ABB RobotStudio station: ExternalGuidedMotion.rsstn

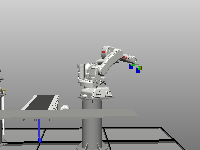
Station E459 (saved by RobotStudio format 3)
Controller NorbertEGMVirtual2, task T_ROB1: task frame (RAPID world) sits at (-305, -752, 720) mm, rotated rx 0 ry 0 rz 30 deg in the station
Controller NorbertEGMVirtual2
  mechanical unit ROB_1: Norbert, 6 joints, base frame (0, 0, 0) mm
  mechanical unit CNV1: ?, 1 joints, base frame (0, 0, 0) mm
Layout (positions relative to the parent item):
  - PedestalR [part, from Libraries\Pedestal.rslib] at (10, 680, 0) mm, rotated rx 0 ry 0 rz 150 deg
  - PedestalN [part, from Libraries\Pedestal.rslib] at (-305, -752, 0) mm, rotated rx 0 ry 0 rz -150 deg
  - Conveyor [part, from Libraries\Conveyor.rslib] at (-998.97, -64.27, 615.81) mm, rotated rx 90 ry 0 rz -90 deg
  - Windowtable [part]
  - BordR [part, from Libraries\Desk.rslib] at (193.4, 1497.66, 0) mm, rotated rx 0 ry 0 rz -120 deg
  - UISpenholder [mechanism, from Libraries\UISpenholder.rslib] at (483.21, 1099.62, 1138) mm, rotated rx -180 ry 0 rz 150 deg
  - Norbert [mechanism, from Robots\IRB140_6_81_C_G_03.rslib] at (-305, -752, 720) mm, rotated rx 0 ry 0 rz 30 deg; joint values [-1.5087, 0.9061, -0.6756, 0, 1.3403, 3.2037] (rad or m)
  - Rudolf [mechanism, from Robots\IRB140_6_81_C_G_03.rslib] at (10, 680, 720) mm, rotated rx 0 ry 0 rz -30 deg; joint values [1.249, 0.6446, -0.2193, 0, 1.1455, 1.249] (rad or m)
  - tSuctionCup [mechanism, from Libraries\tSuctionCup.rslib] at (94.83, -1354.75, 1142.25) mm, rotated rx -180 ry 0 rz -60 deg
Attachment: BordR is attached to PedestalR
Attachment: UISpenholder is attached to Rudolf / Link6
Attachment: tSuctionCup is attached to Norbert / Link6
Station signals: DI doClose, DI doOpen
Station logic (signal -> signal, property => property):
  NorbertEGMVirtual2.doOpen -> SC_Gripper.diOpen
  NorbertEGMVirtual2.doClose -> SC_Gripper.diClose
  SC_Gripper.doClosed -> NorbertEGMVirtual2.diClosed
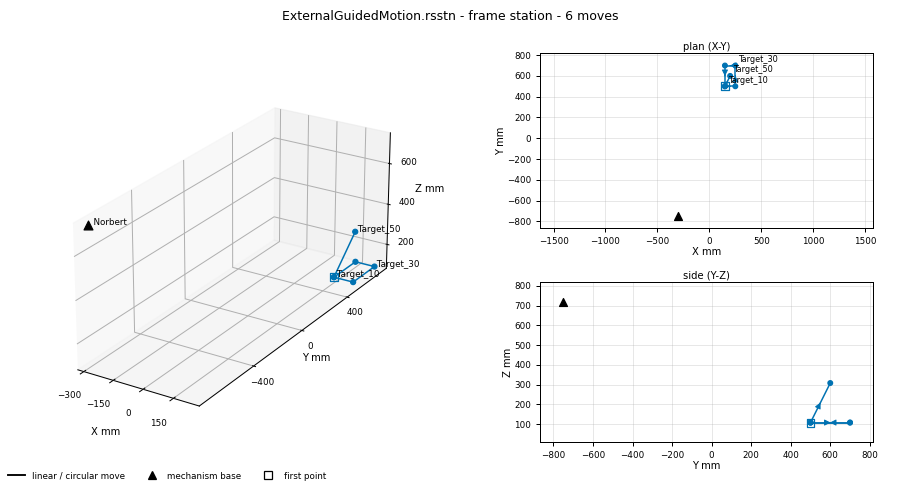
[picture p0: tool path of ExternalGuidedMotion.rsstn in frame station, 6 of 6 moves have a stored position in this frame; points joined in program order, loops and branches not executed]
Targets, tools, work objects and paths stored in the station, written as RAPID:
! task T_ROB1
MODULE CalibData
  PERS tooldata tSuctionCup:=[TRUE,[[120,0,57],[1,0,0,0]],[1,[0,0,1],[1,0,0,0],0,0,0]];
ENDMODULE

! task T_ROB1
MODULE E459RPennTest
  TASK PERS wobjdata wobjBordR:=[FALSE,TRUE,"",[[0,0,0],[1,0,0,0]],[[150,500,8],[1,0,0,0]]];
  CONST robtarget Target_10:=[[0,0,100],[0,0,1,0],[0,0,0,0],[9E9,9E9,9E9,9E9,9E9,9E9]];
  CONST robtarget Target_20:=[[100,0,100],[0,0,1,0],[0,0,0,0],[9E9,9E9,9E9,9E9,9E9,9E9]];
  CONST robtarget Target_30:=[[100,200,100],[0,0,1,0],[0,0,0,0],[9E9,9E9,9E9,9E9,9E9,9E9]];
  CONST robtarget Target_40:=[[0,200,100],[0,0,1,0],[0,0,0,0],[9E9,9E9,9E9,9E9,9E9,9E9]];
  CONST robtarget Target_50:=[[50,100,300],[0,0,1,0],[0,0,0,0],[9E9,9E9,9E9,9E9,9E9,9E9]];
  PROC main()
    Path_10;
  ENDPROC
  PROC Path_10()
    MoveL Target_10,v100,z10,tEnkelPenn\WObj:=wobjBordR;
    MoveL Target_20,v50,z10,tEnkelPenn\WObj:=wobjBordR;
    MoveL Target_30,v100,z10,tEnkelPenn\WObj:=wobjBordR;
    MoveL Target_40,v50,z10,tEnkelPenn\WObj:=wobjBordR;
    MoveL Target_10,v100,z10,tEnkelPenn\WObj:=wobjBordR;
    MoveL Target_50,v100,fine,tEnkelPenn\WObj:=wobjBordR;
  ENDPROC
ENDMODULE

! task T_ROB1
MODULE EnkelPenn
  PERS tooldata tEnkelPenn:=[TRUE,[[0,0,110],[1,0,0,0]],[1,[0,0,1],[1,0,0,0],0,0,0]];
ENDMODULE

